TYPE ST_CrucibleLiftSys :
STRUCT
END_STRUCT
END_TYPE

(* stored: Version 1.1.0.1, ProductVersion 3.1.4024.12
   DUT ST_CrucibleLiftSys: Id {a3be426f-71b1-4854-b3c4-4868d83225ce} *)
